(* IEC 61131-3 sources: cc_kush_rewrite/Functions/Modbus, 13 files *)

(* ---- FC_ModbusReadBool.st ---- *)
// Чтение BOOL из бита Modbus регистра
// Возвращает TRUE при успешном чтении, FALSE при ошибке (неверный индекс бита)
FUNCTION FC_ModbusReadBool : BOOL
VAR_INPUT
    pRegisters : POINTER TO WORD;  // Указатель на массив Modbus регистров
    iRegisterIndex : INT;           // Индекс регистра
    iBitIndex : INT;                // Номер бита в регистре (0..15)
END_VAR
VAR_OUTPUT
    xValue : BOOL;                  // Прочитанное значение
END_VAR
VAR
    wMask : WORD;
    pTargetRegister : POINTER TO WORD;
END_VAR
    // Проверка диапазона индекса бита
    IF iBitIndex >= 0 AND iBitIndex <= 15 THEN
        // Вычислить адрес целевого регистра
        pTargetRegister := pRegisters + iRegisterIndex*2;

        // Создать маску для бита
        wMask := SHL(1, iBitIndex);

        // Прочитать бит
        xValue := (pTargetRegister^ AND wMask) <> 0;

        FC_ModbusReadBool := TRUE;  // Успех
    ELSE
        xValue := FALSE;
        FC_ModbusReadBool := FALSE;  // Ошибка: неверный индекс бита
    END_IF

END_FUNCTION

(* ---- FC_ModbusReadDint.st ---- *)
// Чтение DINT из Modbus регистра
// Возвращает TRUE при успешном чтении
FUNCTION FC_ModbusReadDint : BOOL
VAR_INPUT
    pRegisters : POINTER TO WORD;  // Указатель на массив Modbus регистров
    iRegisterIndex : INT;           // Индекс регистра
END_VAR
VAR_OUTPUT
    iValue : DINT;                   // Прочитанное значение
END_VAR
VAR
    pTargetRegister : POINTER TO WORD;
END_VAR
    // Вычислить адрес целевого регистра и прочитать значение
    pTargetRegister := pRegisters + iRegisterIndex*2;
    iValue := WORD_TO_DINT(pTargetRegister^);
    FC_ModbusReadInt := TRUE;

END_FUNCTION

(* ---- FC_ModbusReadInt.st ---- *)
// Чтение INT из Modbus регистра
// Возвращает TRUE при успешном чтении
FUNCTION FC_ModbusReadInt : BOOL
VAR_INPUT
    pRegisters : POINTER TO WORD;  // Указатель на массив Modbus регистров
    iRegisterIndex : INT;           // Индекс регистра
END_VAR
VAR_OUTPUT
    iValue : INT;                   // Прочитанное значение
END_VAR
VAR
    pTargetRegister : POINTER TO WORD;
END_VAR
    // Вычислить адрес целевого регистра и прочитать значение
    pTargetRegister := pRegisters + iRegisterIndex*2;
    iValue := WORD_TO_INT(pTargetRegister^);
    FC_ModbusReadInt := TRUE;

END_FUNCTION

(* ---- FC_ModbusReadReal.st ---- *)
// Чтение REAL из 2 последовательных Modbus регистров через UNION
// Возвращает TRUE при успешном чтении
// REAL (32 бита) читается из 2 регистров (по 16 бит каждый)
FUNCTION FC_ModbusReadReal : BOOL
VAR_INPUT
    pRegisters : POINTER TO WORD;  // Указатель на массив Modbus регистров
    iRegisterIndex : INT;           // Начальный индекс (читает 2 регистра: N и N+1)
END_VAR
VAR_OUTPUT
    rValue : REAL;                  // Прочитанное значение
END_VAR
VAR
    uConverter : U_RealToWord;
    pTargetRegister : POINTER TO WORD;
END_VAR
    // Чтение первого регистра (младшее слово)
    pTargetRegister := pRegisters + iRegisterIndex*2;
    uConverter.wTag[1] := pTargetRegister^;

    // Чтение второго регистра (старшее слово)
    pTargetRegister := pTargetRegister + 2;
    uConverter.wTag[0] := pTargetRegister^;

    // Преобразовать в REAL
    rValue := uConverter.rTag;

    FC_ModbusReadReal := TRUE;

END_FUNCTION

(* ---- FC_ModbusReadTime.st ---- *)
// Чтение TIME из 2 последовательных Modbus регистров через UNION
// Возвращает TRUE при успешном чтении
// TIME (32 бита) читается из 2 регистров (по 16 бит каждый)
FUNCTION FC_ModbusReadTime : BOOL
VAR_INPUT
    pRegisters : POINTER TO WORD;  // Указатель на массив Modbus регистров
    iRegisterIndex : INT;           // Начальный индекс (читает 2 регистра: N и N+1)
END_VAR
VAR_OUTPUT
    tValue : TIME;                  // Прочитанное значение
END_VAR
VAR
    uConverter : U_TimeToWord;
    pTargetRegister : POINTER TO WORD;
END_VAR
    // Чтение первого регистра (младшее слово)
    pTargetRegister := pRegisters + iRegisterIndex*2;
    uConverter.wTag[1] := pTargetRegister^;

    // Чтение второго регистра (старшее слово)
    pTargetRegister := pTargetRegister + 2;
    uConverter.wTag[0] := pTargetRegister^;

    // Преобразовать в TIME
    tValue := uConverter.tTag;

    FC_ModbusReadTime := TRUE;

END_FUNCTION

(* ---- FC_ModbusReadUdint.st ---- *)
// Чтение UDINT из 2 последовательных Modbus регистров через UNION
// Возвращает TRUE при успешном чтении
// UDINT (32 бита) читается из 2 регистров (по 16 бит каждый)
FUNCTION FC_ModbusReadUdint : BOOL
VAR_INPUT
    pRegisters : POINTER TO WORD;  // Указатель на массив Modbus регистров
    iRegisterIndex : INT;           // Начальный индекс (читает 2 регистра: N и N+1)
END_VAR
VAR_OUTPUT
    udiValue : UDINT;               // Прочитанное значение
END_VAR
VAR
    uConverter : U_UdintToWord;
    pTargetRegister : POINTER TO WORD;
END_VAR
    // Чтение первого регистра (младшее слово)
    pTargetRegister := pRegisters + iRegisterIndex*2;
    uConverter.wTag[1] := pTargetRegister^;

    // Чтение второго регистра (старшее слово)
    pTargetRegister := pTargetRegister + 2;
    uConverter.wTag[0] := pTargetRegister^;

    // Преобразовать в UDINT
    udiValue := uConverter.udiTag;

    FC_ModbusReadUdint := TRUE;

END_FUNCTION

(* ---- FC_ModbusWriteBool.st ---- *)
// Запись BOOL в бит Modbus регистра
// Возвращает TRUE при успешной записи, FALSE при ошибке (неверный индекс бита)
FUNCTION FC_ModbusWriteBool : BOOL
VAR_INPUT
    pRegisters : POINTER TO WORD;  // Указатель на массив Modbus регистров
    iRegisterIndex : INT;           // Индекс регистра
    iBitIndex : INT;                // Номер бита в регистре (0..15)
    xValue : BOOL;                  // Значение для записи
END_VAR
VAR
    wMask : WORD;
    pTargetRegister : POINTER TO WORD;
END_VAR
    // Проверка диапазона индекса бита
    IF iBitIndex >= 0 AND iBitIndex <= 15 THEN
        // Вычислить адрес целевого регистра
        pTargetRegister := pRegisters + iRegisterIndex*2;

        wMask := SHL(1, iBitIndex);  // Создать маску для бита

        IF xValue THEN
            // Установить бит (OR)
            pTargetRegister^ := pTargetRegister^ OR wMask;
        ELSE
            // Сбросить бит (AND NOT)
            pTargetRegister^ := pTargetRegister^ AND NOT wMask;
        END_IF

        FC_ModbusWriteBool := TRUE;  // Успех
    ELSE
        FC_ModbusWriteBool := FALSE;  // Ошибка: неверный индекс бита
    END_IF

END_FUNCTION

(* ---- FC_ModbusWriteDint.st ---- *)
// Запись DINT в 2 последовательных Modbus регистра через UNION
// Возвращает TRUE при успешной записи
// DINT (32 бита) записывается в 2 регистра (по 16 бит каждый)
FUNCTION FC_ModbusWriteDint : BOOL
VAR_INPUT
    pRegisters : POINTER TO WORD;  // Указатель на массив Modbus регистров
    iRegisterIndex : INT;           // Начальный индекс (записывает 2 регистра: N и N+1)
    diValue : DINT;                 // Значение для записи
END_VAR
VAR
    uConverter : U_DintToWord;
    pTargetRegister : POINTER TO WORD;
END_VAR
    // Преобразовать DINT в массив WORD
    uConverter.diTag := diValue;

    // Запись первого регистра (младшее слово)
    pTargetRegister := pRegisters + iRegisterIndex*2;
    pTargetRegister^ := uConverter.wTag[1];

    // Запись второго регистра (старшее слово)
    pTargetRegister := pTargetRegister + 2;
    pTargetRegister^ := uConverter.wTag[0];

    FC_ModbusWriteDint := TRUE;

END_FUNCTION

(* ---- FC_ModbusWriteInt.st ---- *)
// Запись INT в Modbus регистр
// Возвращает TRUE при успешной записи
FUNCTION FC_ModbusWriteInt : BOOL
VAR_INPUT
    pRegisters : POINTER TO WORD;  // Указатель на массив Modbus регистров
    iRegisterIndex : INT;           // Индекс регистра
    iValue : INT;                   // Значение для записи
END_VAR
VAR
    pTargetRegister : POINTER TO WORD;
END_VAR
    // Вычислить адрес целевого регистра и записать значение
    pTargetRegister := pRegisters + iRegisterIndex*2;
    pTargetRegister^ := INT_TO_WORD(iValue);
    FC_ModbusWriteInt := TRUE;

END_FUNCTION

(* ---- FC_ModbusWriteReal.st ---- *)
// Запись REAL в 2 последовательных Modbus регистра через UNION
// Возвращает TRUE при успешной записи
// REAL (32 бита) упаковывается в 2 регистра (по 16 бит каждый)
FUNCTION FC_ModbusWriteReal : BOOL
VAR_INPUT
    pRegisters : POINTER TO WORD;  // Указатель на массив Modbus регистров
    iRegisterIndex : INT;           // Начальный индекс (занимает 2 регистра: N и N+1)
    rValue : REAL;                  // Значение для записи
END_VAR
VAR
    uConverter : U_RealToWord;
    pTargetRegister : POINTER TO WORD;
END_VAR
    uConverter.rTag := rValue;

    // Запись первого регистра (младшее слово)
    pTargetRegister := pRegisters + iRegisterIndex*2;
    pTargetRegister^:= uConverter.wTag[1];

    // Запись второго регистра (старшее слово)
    pTargetRegister := pTargetRegister + 2;
    pTargetRegister^ := uConverter.wTag[0];

    FC_ModbusWriteReal := TRUE;

END_FUNCTION

(* ---- FC_ModbusWriteTime.st ---- *)
// Запись TIME в 2 последовательных Modbus регистра через UNION
// Возвращает TRUE при успешной записи
// TIME (32 бита) упаковывается в 2 регистра (по 16 бит каждый)
FUNCTION FC_ModbusWriteTime : BOOL
VAR_INPUT
    pRegisters : POINTER TO WORD;  // Указатель на массив Modbus регистров
    iRegisterIndex : INT;           // Начальный индекс (занимает 2 регистра: N и N+1)
    tValue : TIME;                  // Значение для записи
END_VAR
VAR
    uConverter : U_TimeToWord;
    pTargetRegister : POINTER TO WORD;
END_VAR
    uConverter.tTag := tValue;

    // Запись первого регистра (младшее слово)
    pTargetRegister := pRegisters + iRegisterIndex*2;
    pTargetRegister^ := uConverter.wTag[1];

    // Запись второго регистра (старшее слово)
    pTargetRegister := pTargetRegister + 2;
    pTargetRegister^ := uConverter.wTag[0];

    FC_ModbusWriteTime := TRUE;

END_FUNCTION

(* ---- FC_ModbusWriteUdint.st ---- *)
// Запись UDINT в 2 последовательных Modbus регистра через UNION
// Возвращает TRUE при успешной записи
// UDINT (32 бита) записывается в 2 регистра (по 16 бит каждый)
FUNCTION FC_ModbusWriteUdint : BOOL
VAR_INPUT
    pRegisters : POINTER TO WORD;  // Указатель на массив Modbus регистров
    iRegisterIndex : INT;           // Начальный индекс (записывает 2 регистра: N и N+1)
    udiValue : UDINT;               // Значение для записи
END_VAR
VAR
    uConverter : U_UdintToWord;
    pTargetRegister : POINTER TO WORD;
END_VAR
    // Преобразовать UDINT в массив WORD
    uConverter.udiTag := udiValue;

    // Запись первого регистра (младшее слово)
    pTargetRegister := pRegisters + iRegisterIndex*2;
    pTargetRegister^ := uConverter.wTag[1];

    // Запись второго регистра (старшее слово)
    pTargetRegister := pTargetRegister + 2;
    pTargetRegister^ := uConverter.wTag[0];

    FC_ModbusWriteUdint := TRUE;

END_FUNCTION

(* ---- FC_ModbusWriteUInt.st ---- *)
FUNCTION FC_ModbusWriteUInt : BOOL
VAR_INPUT
    pRegisters : POINTER TO WORD;  // Указатель на массив Modbus регистров
    iRegisterIndex : INT;           // Индекс регистра
    uValue : UINT;                  // Значение для записи (UINT или enumeration)
END_VAR
VAR
    pTargetRegister : POINTER TO WORD;
END_VAR
    // Вычислить адрес целевого регистра и записать значение
    pTargetRegister := pRegisters + iRegisterIndex*2;
    pTargetRegister^ := UINT_TO_WORD(uValue);
    FC_ModbusWriteUInt := TRUE;

END_FUNCTION
